// TIA Portal V19 export
TYPE "LAF_typeSequenceInterface"
// Interface to control sequence from an HMI
// stored: Access Published
   STRUCT
      commands : "LAF_typeSequenceCommands";
      monitoring { ExternalWritable := 'False'} : "LAF_typeSequenceStatus";
   END_STRUCT;
END_TYPE
